Yaskawa INFORM job: TIMER.JBI

/JOB
//NAME TIMER
//POS
///NPOS 0,0,0,0,0,0
//INST
///DATE 2018/09/11 14:23
///ATTR SC,RW
///GROUP1 RB1,BS1
NOP
TIMER T=600.00
END
